FUNCTION_BLOCK IScISecData (* Composite Function Block Type *)
  (* Standard: 61499-2 *)
  (* Version 0.0, 6/13/2026, Schneider Electric, template *)
  PACKAGE SE.Nereda;
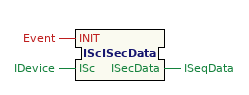
  EVENT_INPUT
    INIT;
  END_EVENT
  SOCKETS
    ISc : IDevice;
  END_SOCKETS
  PLUGS
    ISecData : ISeqData(ServiceAvaiable := TRUE);
  END_PLUGS
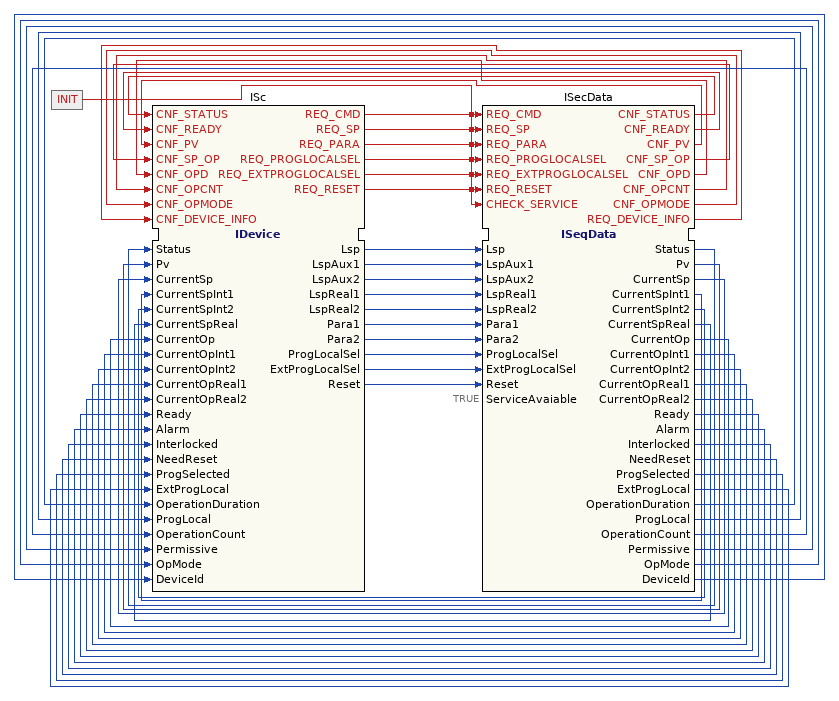
  EVENT_CONNECTIONS
    ISc.REQ_CMD TO ISecData.REQ_CMD;
    ISc.REQ_SP TO ISecData.REQ_SP;
    ISc.REQ_PARA TO ISecData.REQ_PARA;
    ISc.REQ_PROGLOCALSEL TO ISecData.REQ_PROGLOCALSEL;
    ISc.REQ_EXTPROGLOCALSEL TO ISecData.REQ_EXTPROGLOCALSEL;
    ISc.REQ_RESET TO ISecData.REQ_RESET;
    INIT TO ISecData.CHECK_SERVICE;
    ISecData.CNF_STATUS TO ISc.CNF_STATUS;
    ISecData.CNF_READY TO ISc.CNF_READY;
    ISecData.CNF_PV TO ISc.CNF_PV;
    ISecData.CNF_SP_OP TO ISc.CNF_SP_OP;
    ISecData.CNF_OPD TO ISc.CNF_OPD;
    ISecData.CNF_OPCNT TO ISc.CNF_OPCNT;
    ISecData.CNF_OPMODE TO ISc.CNF_OPMODE;
    ISecData.REQ_DEVICE_INFO TO ISc.CNF_DEVICE_INFO;
    INIT TO ISecData.REQ_PARA;
    INIT TO ISecData.REQ_PROGLOCALSEL;
    INIT TO ISecData.REQ_EXTPROGLOCALSEL;
    INIT TO ISecData.REQ_RESET;
    INIT TO ISecData.REQ_CMD;
    INIT TO ISecData.REQ_SP;
  END_CONNECTIONS
  DATA_CONNECTIONS
    ISc.Lsp TO ISecData.Lsp;
    ISc.LspAux1 TO ISecData.LspAux1;
    ISc.LspAux2 TO ISecData.LspAux2;
    ISc.LspReal1 TO ISecData.LspReal1;
    ISc.LspReal2 TO ISecData.LspReal2;
    ISc.Para1 TO ISecData.Para1;
    ISc.Para2 TO ISecData.Para2;
    ISc.ProgLocalSel TO ISecData.ProgLocalSel;
    ISc.ExtProgLocalSel TO ISecData.ExtProgLocalSel;
    ISc.Reset TO ISecData.Reset;
    ISecData.Status TO ISc.Status;
    ISecData.Pv TO ISc.Pv;
    ISecData.CurrentSp TO ISc.CurrentSp;
    ISecData.CurrentSpInt1 TO ISc.CurrentSpInt1;
    ISecData.CurrentSpInt2 TO ISc.CurrentSpInt2;
    ISecData.CurrentSpReal TO ISc.CurrentSpReal;
    ISecData.CurrentOp TO ISc.CurrentOp;
    ISecData.CurrentOpInt1 TO ISc.CurrentOpInt1;
    ISecData.CurrentOpInt2 TO ISc.CurrentOpInt2;
    ISecData.CurrentOpReal1 TO ISc.CurrentOpReal1;
    ISecData.CurrentOpReal2 TO ISc.CurrentOpReal2;
    ISecData.Ready TO ISc.Ready;
    ISecData.Alarm TO ISc.Alarm;
    ISecData.Interlocked TO ISc.Interlocked;
    ISecData.NeedReset TO ISc.NeedReset;
    ISecData.ProgSelected TO ISc.ProgSelected;
    ISecData.ExtProgLocal TO ISc.ExtProgLocal;
    ISecData.OperationDuration TO ISc.OperationDuration;
    ISecData.ProgLocal TO ISc.ProgLocal;
    ISecData.OperationCount TO ISc.OperationCount;
    ISecData.Permissive TO ISc.Permissive;
    ISecData.OpMode TO ISc.OpMode;
    ISecData.DeviceId TO ISc.DeviceId;
  END_CONNECTIONS
END_FUNCTION_BLOCK
